FUNCTION F_WeightCalcByReference : real
VAR_INPUT
	candle	: REFERENCE TO ST_Candle;
END_VAR
VAR
END_VAR

IF candle.dia = 0 THEN
	RETURN;
END_IF

candle.weight := candle.dia*pi*candle.height;

END_FUNCTION

(* stored: Version 1.1.0.1, ProductVersion 3.1.4024.12
   POU F_WeightCalcByReference: Id {34a29e32-8506-4957-8208-2f8d1324afa5}, SpecialFunc None *)
